{attribute 'qualified_only'}
VAR_GLOBAL CONSTANT
	Buffer_Size : INT := 12;
END_VAR

(* stored: Version 1.1.0.1, ProductVersion 3.1.4024.12
   GVL GVL: Id {dce89b43-af45-40e1-bb5c-bcb98d945e8c} *)
